PROGRAM TEST_CYLINDER
VAR
	cylBlock : CylinderBlockBase;
	state : INT;
END_VAR

END_PROGRAM

(* stored: Version 1.1.0.1, ProductVersion 3.1.4020.12
   POU TEST_CYLINDER: Id {9ae041d2-c241-42ec-9562-72f082a519e8}, SpecialFunc None *)
